{attribute 'qualified_only'}
{attribute 'strict'}
TYPE EFeedbackMsgStd900 :
(
	PositionMsg := 10
);
END_TYPE

(* stored: Version 1.1.0.1, ProductVersion 3.1.4024.12
   DUT EFeedbackMsgStd900: Id {1be7c18c-2ca2-4c6d-86ee-0a7c06d3df5c} *)
